// TIA Portal V17 export
// export: Created 2025-03-13T10:30:27.9616027Z, ExportSetting WithDefaults, DisplayName Totally Integrated Automation Portal, DisplayVersion V17 Update 8, DisplayName TIA Portal Openness, DisplayVersion V17 Update 8, DisplayName TIA Portal Version Control Interface, DisplayVersion V17, DisplayName SINAMICS Startdrive Advanced, DisplayVersion V17 SP2, DisplayName SINAMICS Startdrive G110M, G120, G120C, G120D, G120P, G115D, DisplayVersion V17 SP2, DisplayName SINAMICS Startdrive G130, G150, S120, S150, SINAMICS MV, S210, DisplayVersion V17 SP2, DisplayName STEP 7 Professional, DisplayVersion V17 Update 8, DisplayName SINUMERIK ONE STEP 7 Toolbox, DisplayVersion V17 Update 12, DisplayName SINUMERIK 840D sl STEP 7 Toolbox, DisplayVersion V17 Update 12, DisplayName STEP 7 Safety, DisplayVersion V17 Update 6, DisplayName WinCC Advanced, DisplayVersion V17 Update 8
FUNCTION "FC16900_ARRAY_TRANSFER" : Void   // FC16900, LAD
{ S7_Optimized_Access := 'TRUE' }
VERSION : 0.1
// stored: AutoNumber false, IsIECCheckEnabled false, SetENOAutomatically false, UDAEnableTagReadback false
   VAR_INPUT
      INPUT_ARRAY : Array[0..99] of Char;
   END_VAR
   VAR_OUTPUT
      OUTPUT_ARRAY : Array[0..63] of Char;
   END_VAR
   VAR_TEMP
      index : Int;
   END_VAR
BEGIN

REGION Network 1 (SCL)
   FOR #index := 0 TO 63 DO
       #OUTPUT_ARRAY[#index] := #INPUT_ARRAY[#index];
   END_FOR;
END_REGION
END_FUNCTION
